(* Logix 5000 project; controller cow Emulate 5570 rev 36.11; software revision 36.00; part 5 of 6 *)
(* tags used below, declared in another part *)
   ClearLog_T : TIMER;
   Cow_SYS_E : System_Data;
   Cow_SYS_F : System_Data;
   E120RPM : Speed_RPM;
   Err_Reset_T : TIMER;
   Logix_Type : DINT;
   SYS_ON : BOOL;
   B3 : INT[50];
   Bin01 : ALIAS FOR rcp_Big_Bin[0];
   Bin02 : ALIAS FOR rcp_Big_Bin[1];
   Bin03 : ALIAS FOR rcp_Big_Bin[2];
   Bin05 : ALIAS FOR rcp_Big_Bin[4];
   Bin06 : ALIAS FOR rcp_Big_Bin[5];
   Bin07 : ALIAS FOR rcp_Big_Bin[6];
   Bin08 : ALIAS FOR rcp_Big_Bin[7];
   Bin09 : ALIAS FOR rcp_Big_Bin[8];
   Bin10 : ALIAS FOR rcp_Big_Bin[9];
   Bin11 : ALIAS FOR rcp_Big_Bin[10];
   Bin12 : ALIAS FOR rcp_Big_Bin[11];
   Bin13 : ALIAS FOR rcp_Big_Bin[12];
   Bin14 : ALIAS FOR rcp_Big_Bin[13];
   Bin15 : ALIAS FOR rcp_Big_Bin[14];
   Bin16 : ALIAS FOR rcp_Big_Bin[15];
   DateTimes : STRING;
   E112 : MotorX;   // B112
   E120 : MotorX;   // B120
   E141 : MotorX;   // B141
   E142 : MotorX;
   E143 : MotorX;
   E144 : MotorX;
   E145 : MotorX;
   E146 : MotorX;
   E147 : MotorX;
   E148 : MotorX;
   E149 : MotorX;
   E14A : MotorX;
   E14B : MotorX;
   E14C : MotorX;
   E14D : MotorX;
   E14E : MotorX;
   E14F : MotorX;
   E14G : MotorX;
   E331 : SCALE_WEIGHT;
   E340 : Valve;
   E351 : Valve;
   E352 : Valve;
   E45A : Air_Hammer;
   E45B : Air_Hammer;
   E45C : Air_Hammer;
   EINV : Inverter;
   F090 : MotorX;
   F124 : MotorX;
   F125 : MotorX;
   F140 : MotorX;
   F167 : MotorX;
   F168 : MotorX;
   F240 : MotorX;
   F270 : MotorX;
   F363 : Branch_SV2;
   F364 : Branch_SV2;
   F413 : MotorX;
   F441 : MotorX;
   F560 : MotorX;
   F561 : MotorX;
   LED_Batch_seq : DINT;
   LED_Batch_Total : ALIAS FOR rcp_Recipe.BatchSet;
   Led_Hand_PartNumber : DINT;
   Led_Hand_RealWeight : REAL;
   LED_Hand_SetWeight : REAL;
   Led_string : STRING[16];
   Now : DateTime_Type;
   rcp_Big_Scale : REAL;
   rcp_Big_Speed : DINT;
   rcp_Hand_Run : BOOL;
   rcp_Recipe : Recipe_Type;
   rcp_ScheduleLog : ScheduleLog[10];
   SCALE_SIMULATE : BOOL;
   STS : INT[100];
   SYS : System_Common;
   SYS_E : Sys_Data;
   SYS_F : Sys_Data;
(* MainProgram, continued *)

ROUTINE Device_E   (* ladder *)
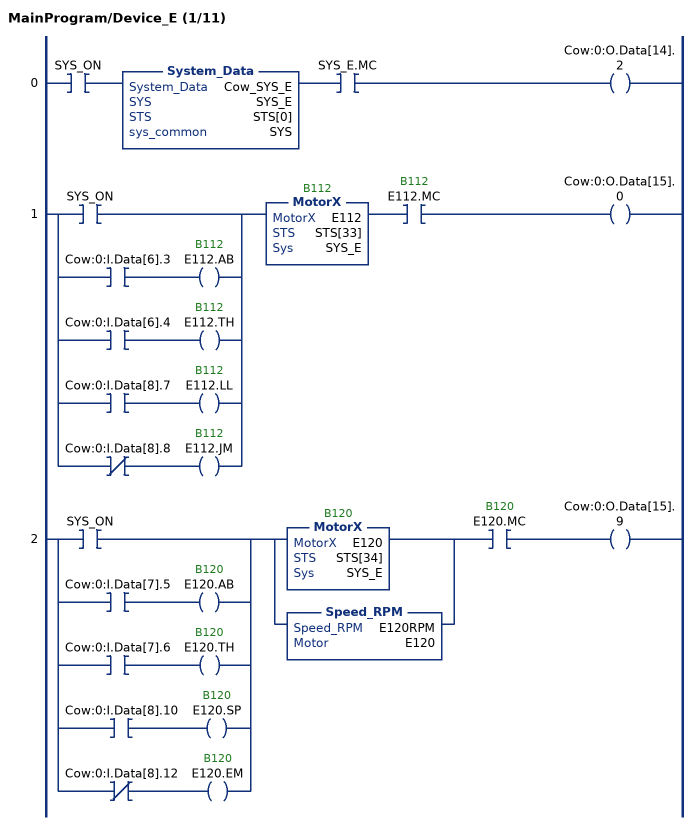
   0: XIC(SYS_ON)System_Data(Cow_SYS_E,SYS_E,STS[0],SYS)XIC(SYS_E.MC)OTE(Cow:0:O.Data[14].2);
   1: [XIC(SYS_ON) ,XIC(Cow:0:I.Data[6].3) OTE(E112.AB) ,XIC(Cow:0:I.Data[6].4) OTE(E112.TH) ,XIC(Cow:0:I.Data[8].7) OTE(E112.LL) ,XIO(Cow:0:I.Data[8].8) OTE(E112.JM) ]MotorX(E112,STS[33],SYS_E)XIC(E112.MC)OTE(Cow:0:O.Data[15].0);
   2: [XIC(SYS_ON) ,XIC(Cow:0:I.Data[7].5) OTE(E120.AB) ,XIC(Cow:0:I.Data[7].6) OTE(E120.TH) ,XIC(Cow:0:I.Data[8].10) OTE(E120.SP) ,XIO(Cow:0:I.Data[8].12) OTE(E120.EM) ][MotorX(E120,STS[34],SYS_E) ,Speed_RPM(E120RPM,E120) ]XIC(E120.MC)OTE(Cow:0:O.Data[15].9);
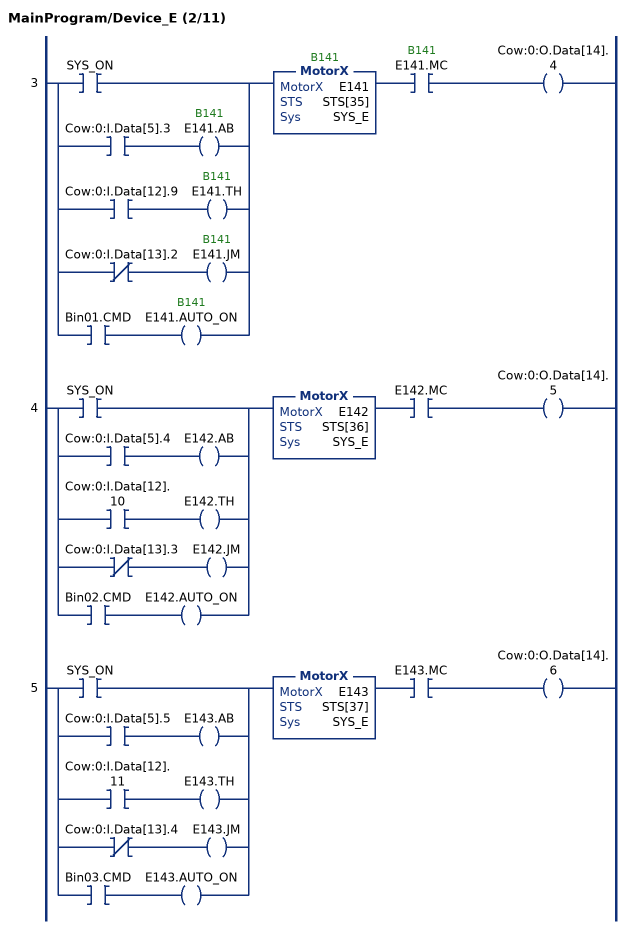
   3: [XIC(SYS_ON) ,XIC(Cow:0:I.Data[5].3) OTE(E141.AB) ,XIC(Cow:0:I.Data[12].9) OTE(E141.TH) ,XIO(Cow:0:I.Data[13].2) OTE(E141.JM) ,XIC(Bin01.CMD) OTE(E141.AUTO_ON) ]MotorX(E141,STS[35],SYS_E)XIC(E141.MC)OTE(Cow:0:O.Data[14].4);
   4: [XIC(SYS_ON) ,XIC(Cow:0:I.Data[5].4) OTE(E142.AB) ,XIC(Cow:0:I.Data[12].10) OTE(E142.TH) ,XIO(Cow:0:I.Data[13].3) OTE(E142.JM) ,XIC(Bin02.CMD) OTE(E142.AUTO_ON) ]MotorX(E142,STS[36],SYS_E)XIC(E142.MC)OTE(Cow:0:O.Data[14].5);
   5: [XIC(SYS_ON) ,XIC(Cow:0:I.Data[5].5) OTE(E143.AB) ,XIC(Cow:0:I.Data[12].11) OTE(E143.TH) ,XIO(Cow:0:I.Data[13].4) OTE(E143.JM) ,XIC(Bin03.CMD) OTE(E143.AUTO_ON) ]MotorX(E143,STS[37],SYS_E)XIC(E143.MC)OTE(Cow:0:O.Data[14].6);
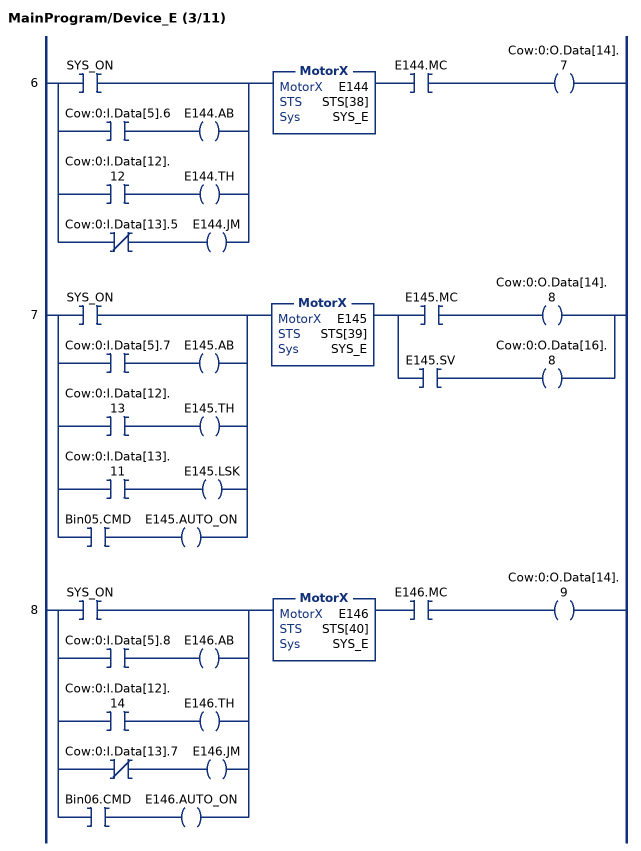
   6: [XIC(SYS_ON) ,XIC(Cow:0:I.Data[5].6) OTE(E144.AB) ,XIC(Cow:0:I.Data[12].12) OTE(E144.TH) ,XIO(Cow:0:I.Data[13].5) OTE(E144.JM) ]MotorX(E144,STS[38],SYS_E)XIC(E144.MC)OTE(Cow:0:O.Data[14].7);
   7: [XIC(SYS_ON) ,XIC(Cow:0:I.Data[5].7) OTE(E145.AB) ,XIC(Cow:0:I.Data[12].13) OTE(E145.TH) ,XIC(Cow:0:I.Data[13].11) OTE(E145.LSK) ,XIC(Bin05.CMD) OTE(E145.AUTO_ON) ]MotorX(E145,STS[39],SYS_E)[XIC(E145.MC) OTE(Cow:0:O.Data[14].8) ,XIC(E145.SV) OTE(Cow:0:O.Data[16].8) ];
   8: [XIC(SYS_ON) ,XIC(Cow:0:I.Data[5].8) OTE(E146.AB) ,XIC(Cow:0:I.Data[12].14) OTE(E146.TH) ,XIO(Cow:0:I.Data[13].7) OTE(E146.JM) ,XIC(Bin06.CMD) OTE(E146.AUTO_ON) ]MotorX(E146,STS[40],SYS_E)XIC(E146.MC)OTE(Cow:0:O.Data[14].9);
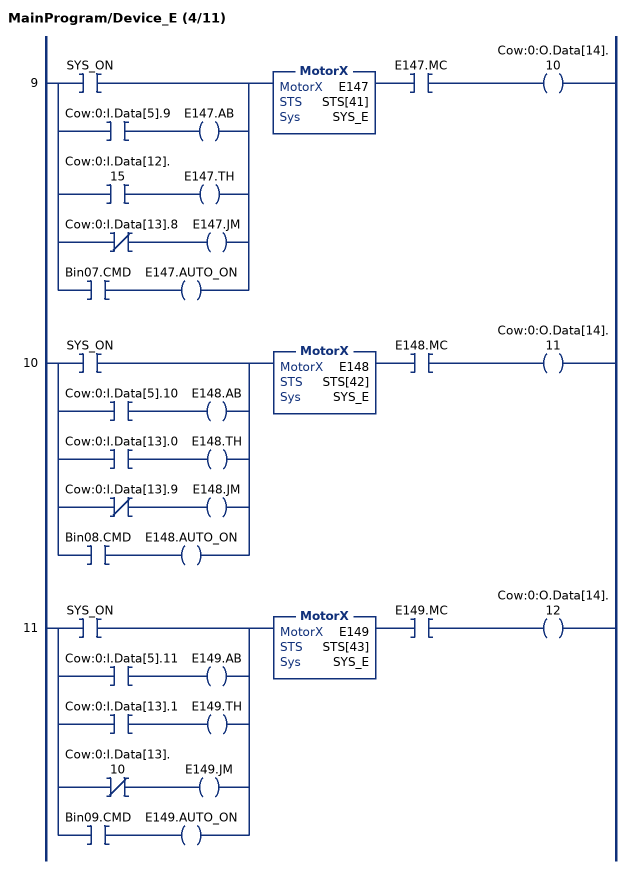
   9: [XIC(SYS_ON) ,XIC(Cow:0:I.Data[5].9) OTE(E147.AB) ,XIC(Cow:0:I.Data[12].15) OTE(E147.TH) ,XIO(Cow:0:I.Data[13].8) OTE(E147.JM) ,XIC(Bin07.CMD) OTE(E147.AUTO_ON) ]MotorX(E147,STS[41],SYS_E)XIC(E147.MC)OTE(Cow:0:O.Data[14].10);
   10: [XIC(SYS_ON) ,XIC(Cow:0:I.Data[5].10) OTE(E148.AB) ,XIC(Cow:0:I.Data[13].0) OTE(E148.TH) ,XIO(Cow:0:I.Data[13].9) OTE(E148.JM) ,XIC(Bin08.CMD) OTE(E148.AUTO_ON) ]MotorX(E148,STS[42],SYS_E)XIC(E148.MC)OTE(Cow:0:O.Data[14].11);
   11: [XIC(SYS_ON) ,XIC(Cow:0:I.Data[5].11) OTE(E149.AB) ,XIC(Cow:0:I.Data[13].1) OTE(E149.TH) ,XIO(Cow:0:I.Data[13].10) OTE(E149.JM) ,XIC(Bin09.CMD) OTE(E149.AUTO_ON) ]MotorX(E149,STS[43],SYS_E)XIC(E149.MC)OTE(Cow:0:O.Data[14].12);
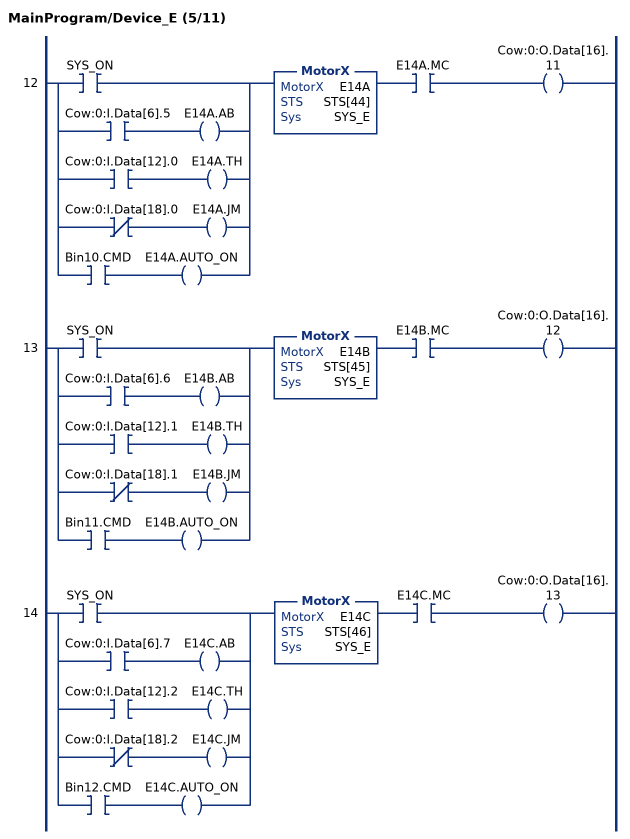
   12: [XIC(SYS_ON) ,XIC(Cow:0:I.Data[6].5) OTE(E14A.AB) ,XIC(Cow:0:I.Data[12].0) OTE(E14A.TH) ,XIO(Cow:0:I.Data[18].0) OTE(E14A.JM) ,XIC(Bin10.CMD) OTE(E14A.AUTO_ON) ]MotorX(E14A,STS[44],SYS_E)XIC(E14A.MC)OTE(Cow:0:O.Data[16].11);
   13: [XIC(SYS_ON) ,XIC(Cow:0:I.Data[6].6) OTE(E14B.AB) ,XIC(Cow:0:I.Data[12].1) OTE(E14B.TH) ,XIO(Cow:0:I.Data[18].1) OTE(E14B.JM) ,XIC(Bin11.CMD) OTE(E14B.AUTO_ON) ]MotorX(E14B,STS[45],SYS_E)XIC(E14B.MC)OTE(Cow:0:O.Data[16].12);
   14: [XIC(SYS_ON) ,XIC(Cow:0:I.Data[6].7) OTE(E14C.AB) ,XIC(Cow:0:I.Data[12].2) OTE(E14C.TH) ,XIO(Cow:0:I.Data[18].2) OTE(E14C.JM) ,XIC(Bin12.CMD) OTE(E14C.AUTO_ON) ]MotorX(E14C,STS[46],SYS_E)XIC(E14C.MC)OTE(Cow:0:O.Data[16].13);
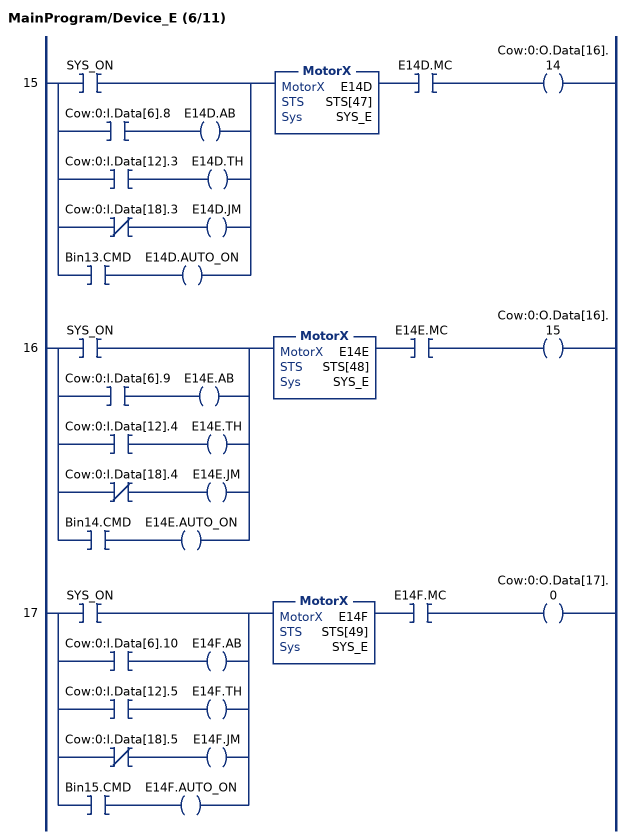
   15: [XIC(SYS_ON) ,XIC(Cow:0:I.Data[6].8) OTE(E14D.AB) ,XIC(Cow:0:I.Data[12].3) OTE(E14D.TH) ,XIO(Cow:0:I.Data[18].3) OTE(E14D.JM) ,XIC(Bin13.CMD) OTE(E14D.AUTO_ON) ]MotorX(E14D,STS[47],SYS_E)XIC(E14D.MC)OTE(Cow:0:O.Data[16].14);
   16: [XIC(SYS_ON) ,XIC(Cow:0:I.Data[6].9) OTE(E14E.AB) ,XIC(Cow:0:I.Data[12].4) OTE(E14E.TH) ,XIO(Cow:0:I.Data[18].4) OTE(E14E.JM) ,XIC(Bin14.CMD) OTE(E14E.AUTO_ON) ]MotorX(E14E,STS[48],SYS_E)XIC(E14E.MC)OTE(Cow:0:O.Data[16].15);
   17: [XIC(SYS_ON) ,XIC(Cow:0:I.Data[6].10) OTE(E14F.AB) ,XIC(Cow:0:I.Data[12].5) OTE(E14F.TH) ,XIO(Cow:0:I.Data[18].5) OTE(E14F.JM) ,XIC(Bin15.CMD) OTE(E14F.AUTO_ON) ]MotorX(E14F,STS[49],SYS_E)XIC(E14F.MC)OTE(Cow:0:O.Data[17].0);
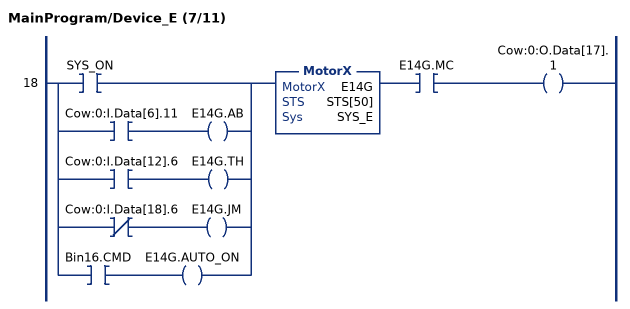
   18: [XIC(SYS_ON) ,XIC(Cow:0:I.Data[6].11) OTE(E14G.AB) ,XIC(Cow:0:I.Data[12].6) OTE(E14G.TH) ,XIO(Cow:0:I.Data[18].6) OTE(E14G.JM) ,XIC(Bin16.CMD) OTE(E14G.AUTO_ON) ]MotorX(E14G,STS[50],SYS_E)XIC(E14G.MC)OTE(Cow:0:O.Data[17].1);
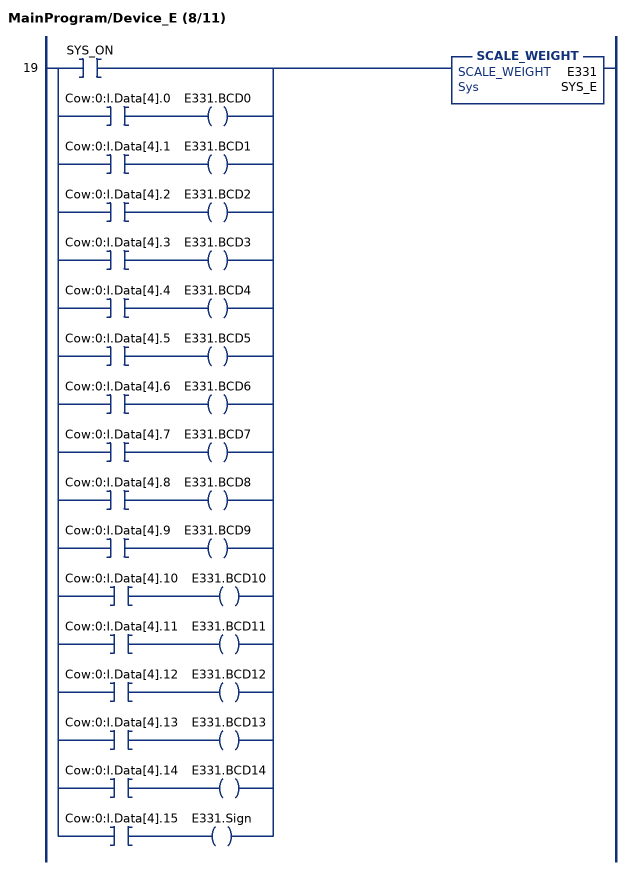
   19: [XIC(SYS_ON) ,XIC(Cow:0:I.Data[4].0) OTE(E331.BCD0) ,XIC(Cow:0:I.Data[4].1) OTE(E331.BCD1) ,XIC(Cow:0:I.Data[4].2) OTE(E331.BCD2) ,XIC(Cow:0:I.Data[4].3) OTE(E331.BCD3) ,XIC(Cow:0:I.Data[4].4) OTE(E331.BCD4) ,XIC(Cow:0:I.Data[4].5) OTE(E331.BCD5) ,XIC(Cow:0:I.Data[4].6) OTE(E331.BCD6) ,XIC(Cow:0:I.Data[4].7) OTE(E331.BCD7) ,XIC(Cow:0:I.Data[4].8) OTE(E331.BCD8) ,XIC(Cow:0:I.Data[4].9) OTE(E331.BCD9) ,XIC(Cow:0:I.Data[4].10) OTE(E331.BCD10) ,XIC(Cow:0:I.Data[4].11) OTE(E331.BCD11) ,XIC(Cow:0:I.Data[4].12) OTE(E331.BCD12) ,XIC(Cow:0:I.Data[4].13) OTE(E331.BCD13) ,XIC(Cow:0:I.Data[4].14) OTE(E331.BCD14) ,XIC(Cow:0:I.Data[4].15) OTE(E331.Sign) ]SCALE_WEIGHT(E331,SYS_E);
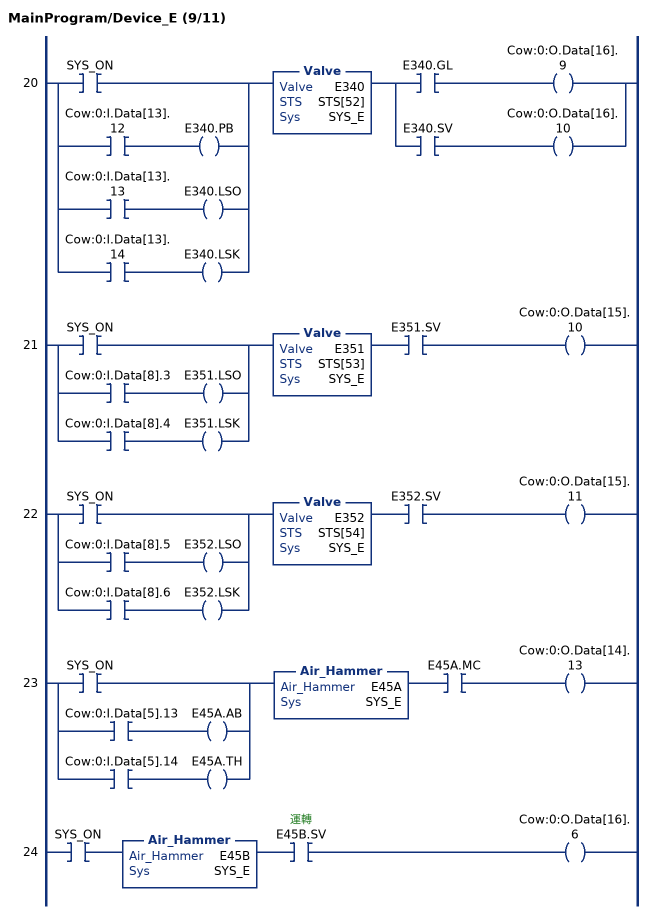
   20: [XIC(SYS_ON) ,XIC(Cow:0:I.Data[13].12) OTE(E340.PB) ,XIC(Cow:0:I.Data[13].13) OTE(E340.LSO) ,XIC(Cow:0:I.Data[13].14) OTE(E340.LSK) ]Valve(E340,STS[52],SYS_E)[XIC(E340.GL) OTE(Cow:0:O.Data[16].9) ,XIC(E340.SV) OTE(Cow:0:O.Data[16].10) ];
   21: [XIC(SYS_ON) ,XIC(Cow:0:I.Data[8].3) OTE(E351.LSO) ,XIC(Cow:0:I.Data[8].4) OTE(E351.LSK) ]Valve(E351,STS[53],SYS_E)XIC(E351.SV)OTE(Cow:0:O.Data[15].10);
   22: [XIC(SYS_ON) ,XIC(Cow:0:I.Data[8].5) OTE(E352.LSO) ,XIC(Cow:0:I.Data[8].6) OTE(E352.LSK) ]Valve(E352,STS[54],SYS_E)XIC(E352.SV)OTE(Cow:0:O.Data[15].11);
   23: [XIC(SYS_ON) ,XIC(Cow:0:I.Data[5].13) OTE(E45A.AB) ,XIC(Cow:0:I.Data[5].14) OTE(E45A.TH) ]Air_Hammer(E45A,SYS_E)XIC(E45A.MC)OTE(Cow:0:O.Data[14].13);
   24: XIC(SYS_ON)Air_Hammer(E45B,SYS_E)XIC(E45B.SV)OTE(Cow:0:O.Data[16].6);
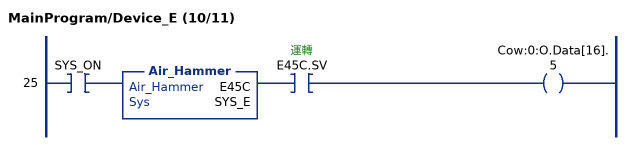
   25: XIC(SYS_ON)Air_Hammer(E45C,SYS_E)XIC(E45C.SV)OTE(Cow:0:O.Data[16].5);
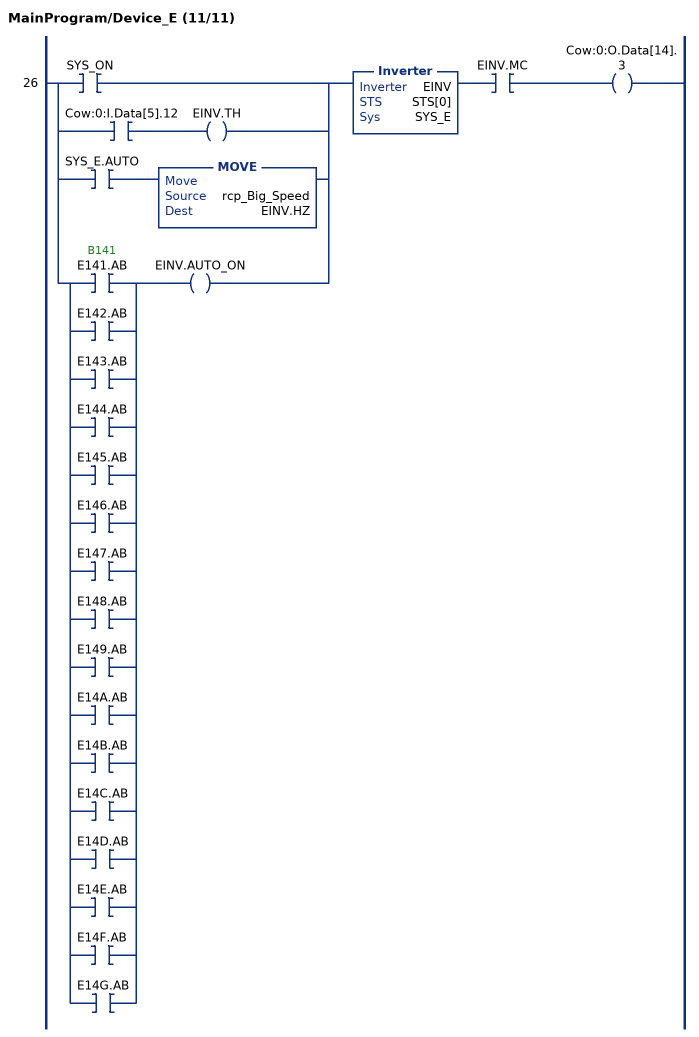
   26: [XIC(SYS_ON) ,XIC(Cow:0:I.Data[5].12) OTE(EINV.TH) ,XIC(SYS_E.AUTO) MOVE(rcp_Big_Speed,EINV.HZ) ,[XIC(E141.AB) ,XIC(E142.AB) ,XIC(E143.AB) ,XIC(E144.AB) ,XIC(E145.AB) ,XIC(E146.AB) ,XIC(E147.AB) ,XIC(E148.AB) ,XIC(E149.AB) ,XIC(E14A.AB) ,XIC(E14B.AB) ,XIC(E14C.AB) ,XIC(E14D.AB) ,XIC(E14E.AB) ,XIC(E14F.AB) ,XIC(E14G.AB) ] OTE(EINV.AUTO_ON) ]Inverter(EINV,STS[0],SYS_E)XIC(EINV.MC)OTE(Cow:0:O.Data[14].3);
END_ROUTINE

ROUTINE Device_F   (* ladder *)
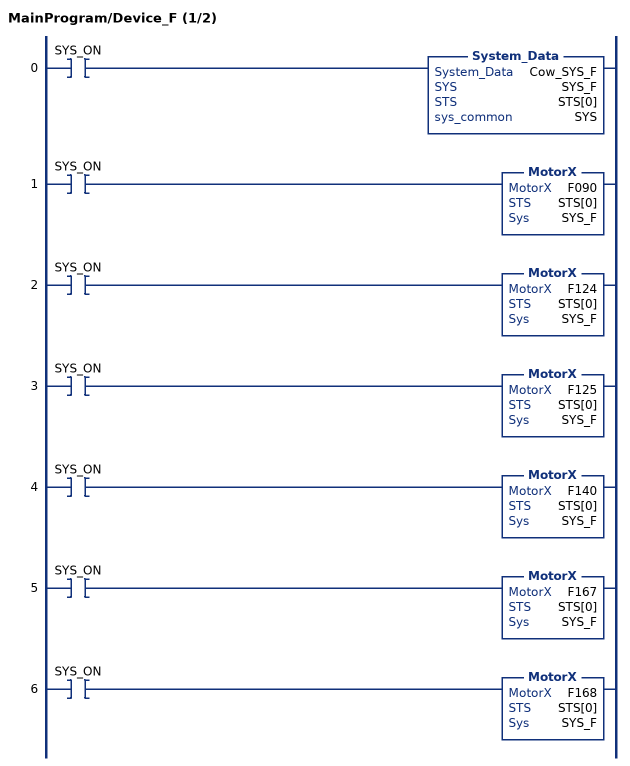
   0: XIC(SYS_ON)System_Data(Cow_SYS_F,SYS_F,STS[0],SYS);
   1: XIC(SYS_ON)MotorX(F090,STS[0],SYS_F);
   2: XIC(SYS_ON)MotorX(F124,STS[0],SYS_F);
   3: XIC(SYS_ON)MotorX(F125,STS[0],SYS_F);
   4: XIC(SYS_ON)MotorX(F140,STS[0],SYS_F);
   5: XIC(SYS_ON)MotorX(F167,STS[0],SYS_F);
   6: XIC(SYS_ON)MotorX(F168,STS[0],SYS_F);
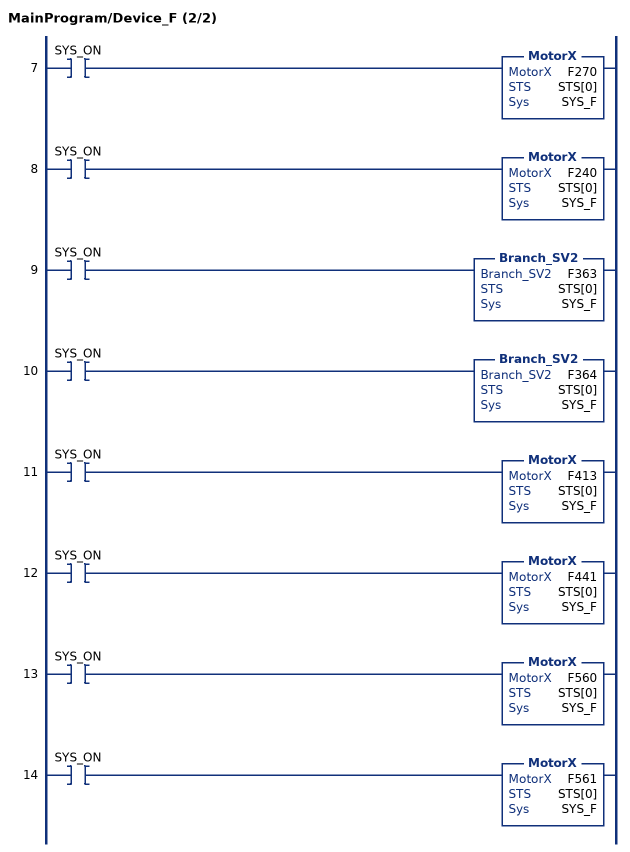
   7: XIC(SYS_ON)MotorX(F270,STS[0],SYS_F);
   8: XIC(SYS_ON)MotorX(F240,STS[0],SYS_F);
   9: XIC(SYS_ON)Branch_SV2(F363,STS[0],SYS_F);
   10: XIC(SYS_ON)Branch_SV2(F364,STS[0],SYS_F);
   11: XIC(SYS_ON)MotorX(F413,STS[0],SYS_F);
   12: XIC(SYS_ON)MotorX(F441,STS[0],SYS_F);
   13: XIC(SYS_ON)MotorX(F560,STS[0],SYS_F);
   14: XIC(SYS_ON)MotorX(F561,STS[0],SYS_F);
END_ROUTINE

ROUTINE MainRoutine   (* ladder *)
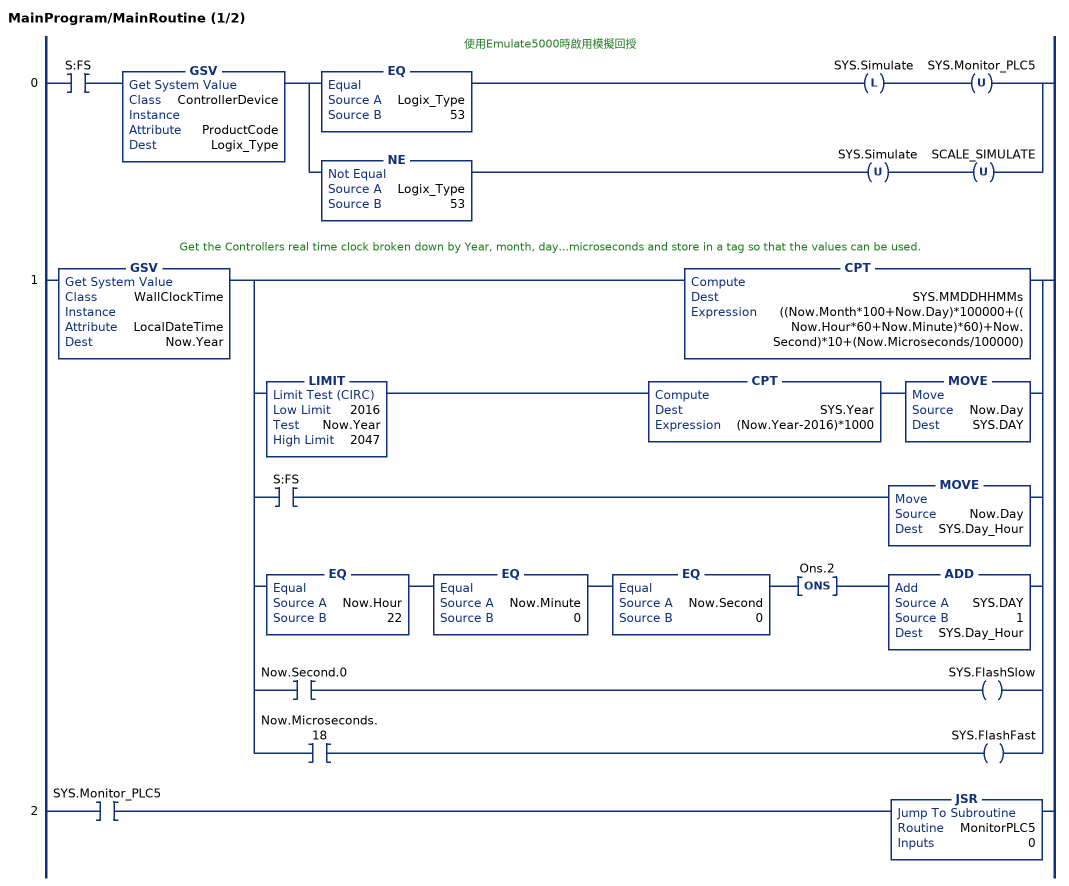
   // 使用Emulate5000時啟用模擬回授
   0: XIC(S:FS)GSV(ControllerDevice,,ProductCode,Logix_Type)[EQ(Logix_Type,53) OTL(SYS.Simulate) OTU(SYS.Monitor_PLC5) ,NE(Logix_Type,53) OTU(SYS.Simulate) OTU(SCALE_SIMULATE) ];
   // Get the Controllers real time clock broken down by Year, month, day...microseconds and store in a tag so that the values can be used.
   1: GSV(WallClockTime,,LocalDateTime,Now.Year)[CPT(SYS.MMDDHHMMs,((Now.Month*100+Now.Day)*100000+((Now.Hour*60+Now.Minute)*60)+Now.Second)*10+(Now.Microseconds/100000)) ,LIMIT(2016,Now.Year,2047) CPT(SYS.Year,(Now.Year-2016)*1000) MOVE(Now.Day,SYS.DAY) ,XIC(S:FS) MOVE(Now.Day,SYS.Day_Hour) ,EQ(Now.Hour,22) EQ(Now.Minute,0) EQ(Now.Second,0) ONS(Ons.2) ADD(SYS.DAY,1,SYS.Day_Hour) ,XIC(Now.Second.0) OTE(SYS.FlashSlow) ,XIC(Now.Microseconds.18) OTE(SYS.FlashFast) ];
   2: XIC(SYS.Monitor_PLC5)JSR(MonitorPLC5,0);
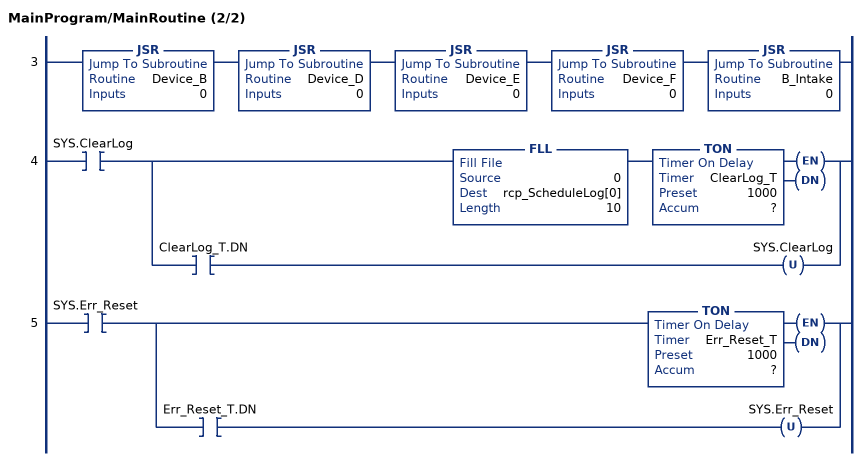
   3: JSR(Device_B,0)JSR(Device_D,0)JSR(Device_E,0)JSR(Device_F,0)JSR(B_Intake,0);
   4: XIC(SYS.ClearLog)[FLL(0,rcp_ScheduleLog[0],10) TON(ClearLog_T,?,?) ,XIC(ClearLog_T.DN) OTU(SYS.ClearLog) ];
   5: XIC(SYS.Err_Reset)[TON(Err_Reset_T,?,?) ,XIC(Err_Reset_T.DN) OTU(SYS.Err_Reset) ];
END_ROUTINE

ROUTINE MonitorPLC5   (* ladder *)
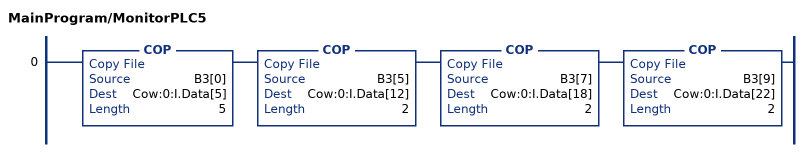
   0: COP(B3[0],Cow:0:I.Data[5],5)COP(B3[5],Cow:0:I.Data[12],2)COP(B3[7],Cow:0:I.Data[18],2)COP(B3[9],Cow:0:I.Data[22],2);
END_ROUTINE
END_PROGRAM

PROGRAM Recipe   (* main routine MainRoutine *)
VAR
   Batch_delay : TIMER := (PRE := 3000, ACC := 3000);
   Big_Add : TIMER := (PRE := 2000, ACC := 2000);
   Big_Avg : REAL := 3.0;
   Big_Bin_Changed : BOOL;
   Big_Bridge_time : TIMER := (PRE := 10000);
   Big_Change_Weight : REAL;
   Big_Error_Over : BOOL;
   Big_ErrorWeight : REAL := 8.0;
   Big_id : DINT;
   Big_id1 : DINT;
   Big_Idx : DINT := 2;
   Big_Index : DINT := 2;
   Big_Prev : REAL;
   Big_Run_Fs : BOOL;
   Big_Scale1 : REAL;
   Big_Scale2 : REAL := 873.0;
   Big_Scale3 : REAL := 882.0;
   Big_Timer : TIMER := (PRE := 3000);
   Big_w : REAL[11] := ([0] := 3.0, [10] := 3.0);
   Big_Weight_Control : CONTROL := (LEN := 10, POS := 1);
   BigBin_Change_ID : DINT := 4;
   Bin_Index : DINT := 1;
   change_cycle : TIMER := (PRE := 200, ACC := 53, EN := 1, TT := 1);
   Find : BOOL;
   Hand_Index : DINT := 1;
   Hand_Scale1 : REAL;
   Index : DINT := 15;
   INDEX1 : DINT := 16;
   Led_Hand_Part : STRING := '0  0.0  0.0';
   Led_Recipe : STRING := 'Test$00$00$00$00$00$00 2-1';
   Led_str : String20[10] := ([0] := '0', [1] := ' 0.0', [2] := ' 0.0', [3] := ' ', [4] := ' ', [5] := 'Test$00$00$00$00$00$00', [6] := ' ', [7] := '2', [8] := '1', [9] := '-');
        [0]   // 手投原料編號
        [1]   // 手投原料設重
        [2]   // 手投原料實重
        [5]   // 配方編號
        [6]   // 空格
        [7]   // 批次
        [8]   // 總批次
   Max_BigID : DINT := 17;
   No_Big_CMD : BOOL := 1;
   Ons : BOOL[64] := ([0] := 1, [1] := 1, [4] := 1, [8] := 1, [9] := 1, [11] := 1, [13] := 1, [15] := 1, [19] := 1, [23] := 1, [24] := 1, [27] := 1, [29] := 1, [31] := 1, [32] := 1, [33] := 1, [35] := 1, [46] := 1, [47] := 1, [59] := 1, [60] := 1, [61] := 1, [62] := 1);
   Part_Index : DINT := 20;
   rcp_Batch_Finish : BOOL;
   rcp_Big1 : Part_Type := (Bin[0] := 1, Bin[1] := 2, Bin_Index[1] := 1, Number[0] := 730000570, Number[1] := 730000930, SetWeight[0] := 300.0, SetWeight[1] := 600.0);
   rcp_Big_Bridge_delay : TIMER := (PRE := 20000);
   rcp_BigBin_Bridge : DINT := 1;
   rcp_BigLastID1 : DINT := 2;
   Recipe_Mult : CONTROL := (LEN := 17);
   Report_TIMER : TIMER := (PRE := 3000);
   RTOS_Hand_WeightReal : RTOS_Format;
   RTOS_Hand_WeightSet : RTOS_Format;
   Scale_Simulate_Timer : TIMER := (PRE := 200, ACC := 53, EN := 1, TT := 1);
   Simulate_Big_w : REAL := 1.0;
   TMP : DINT;
   ZERO : DINT[100];
END_VAR

ROUTINE Average_weight   (* ladder *)
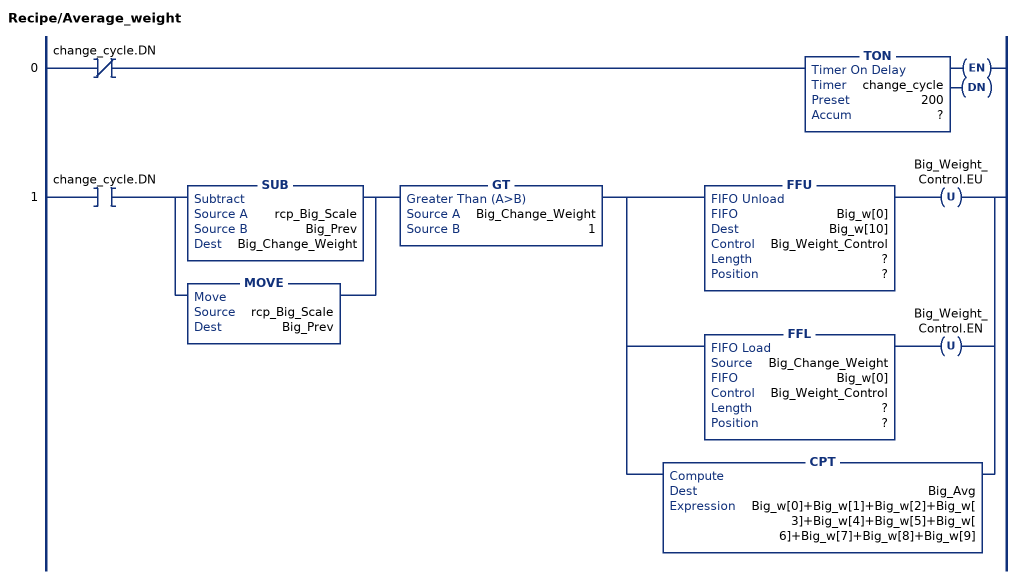
   0: XIO(change_cycle.DN)TON(change_cycle,?,?);
   1: XIC(change_cycle.DN)[SUB(rcp_Big_Scale,Big_Prev,Big_Change_Weight) ,MOVE(rcp_Big_Scale,Big_Prev) ]GT(Big_Change_Weight,1)[FFU(Big_w[0],Big_w[10],Big_Weight_Control,?,?) OTU(Big_Weight_Control.EU) ,FFL(Big_Change_Weight,Big_w[0],Big_Weight_Control,?,?) OTU(Big_Weight_Control.EN) ,CPT(Big_Avg,Big_w[0]+Big_w[1]+Big_w[2]+Big_w[3]+Big_w[4]+Big_w[5]+Big_w[6]+Big_w[7]+Big_w[8]+Big_w[9]) ];
END_ROUTINE

ROUTINE LED   (* ladder *)
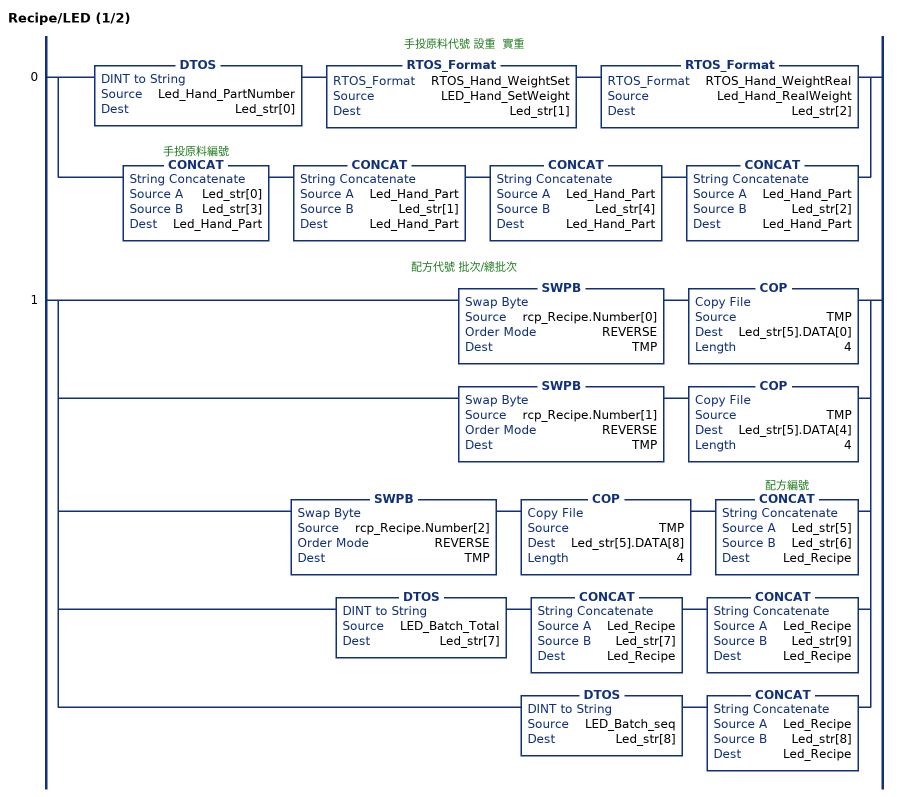
   // 手投原料代號 設重  實重
   0: [DTOS(Led_Hand_PartNumber,Led_str[0]) RTOS_Format(RTOS_Hand_WeightSet,LED_Hand_SetWeight,Led_str[1]) RTOS_Format(RTOS_Hand_WeightReal,Led_Hand_RealWeight,Led_str[2]) ,CONCAT(Led_str[0],Led_str[3],Led_Hand_Part) CONCAT(Led_Hand_Part,Led_str[1],Led_Hand_Part) CONCAT(Led_Hand_Part,Led_str[4],Led_Hand_Part) CONCAT(Led_Hand_Part,Led_str[2],Led_Hand_Part) ];
   // 配方代號 批次/總批次
   1: [SWPB(rcp_Recipe.Number[0],REVERSE,TMP) COP(TMP,Led_str[5].DATA[0],4) ,SWPB(rcp_Recipe.Number[1],REVERSE,TMP) COP(TMP,Led_str[5].DATA[4],4) ,SWPB(rcp_Recipe.Number[2],REVERSE,TMP) COP(TMP,Led_str[5].DATA[8],4) CONCAT(Led_str[5],Led_str[6],Led_Recipe) ,DTOS(LED_Batch_Total,Led_str[7]) CONCAT(Led_Recipe,Led_str[7],Led_Recipe) CONCAT(Led_Recipe,Led_str[9],Led_Recipe) ,DTOS(LED_Batch_seq,Led_str[8]) CONCAT(Led_Recipe,Led_str[8],Led_Recipe) ];
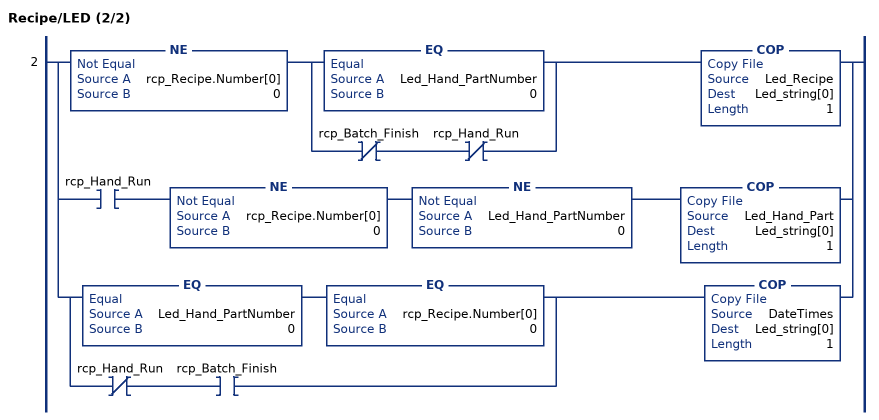
   2: [NE(rcp_Recipe.Number[0],0) [EQ(Led_Hand_PartNumber,0) ,XIO(rcp_Batch_Finish) XIO(rcp_Hand_Run) ] COP(Led_Recipe,Led_string[0],1) ,XIC(rcp_Hand_Run) NE(rcp_Recipe.Number[0],0) NE(Led_Hand_PartNumber,0) COP(Led_Hand_Part,Led_string[0],1) ,[EQ(Led_Hand_PartNumber,0) EQ(rcp_Recipe.Number[0],0) ,XIO(rcp_Hand_Run) XIC(rcp_Batch_Finish) ] COP(DateTimes,Led_string[0],1) ];
END_ROUTINE
